FB_ECAT_DIAG(
	nEcMasterSlaveCount:= , 
	nEcMasterDevState:= , 
	nEcMasterDeviceId:= , 
	arrEcMasterNetId:= , 
	nEcMasterSlaveCountCfg:= , 
	wFrmXWcState:= , 
	bAllFrameWcStatesOK=> , 
	bEtherCATOK=> , 
	bFrameWcStateError=> , 
	bSlaveCountError=> , 
	bMasterDevStateError=> , 
	stMasterDevState=> , 
	bBusy=> , 
	bError=> , 
	iErrorID=> , 
	arrSlaveInfo:= arrEcatSlaveInfo);

IF nSlaveNr > iSLAVEADDR_ARR_SIZE THEN nSlaveNr := iSLAVEADDR_ARR_SIZE; END_IF
stSlaveInfo := arrEcatSlaveInfo[nSlaveNr];


FB_EVENTHANDLER(
	bClearAll:= bAckP, 
	bAlarmActive=> , 
	sEventText=> , 
	sEventSource=> , 
	sEventJson=> );

END_PROGRAM

// ---- POUs/MesTest.TcPOU
PROGRAM MesTest
VAR
	MES:						FB_MES_INTERFACE_V2;		(* Instance of MES-Interface function block *)
	bMES_InitOK					:BOOL := FALSE;
	RESP:						ST_REQUEST;				(* Reference to MES-Interface function block response *)
	RESET:						BOOL;					
	START:						BOOL;					
	STATE:						UDINT;
	INDEX:						INT;					
	
	COVER_BARCODE:				STRING:='288000060010020103725571';					(* COVER barcode *)
	COVER_PARENT:				STRING;					(* MRT parent barcode *)
	COVER_STATE:				ST_GET_OP_STATE;		(* Container of SFC State data which releated to Cover barcode *)
	COVER_INVENTORY:			ST_INVENTORY;			(* Result inventory of the import *)
	COVER_VALID:				BOOL;					
	
	CARRIER_BARCODE:			STRING:='288000000005020103725189';					(* CARRIER barcode *)
	CARRIER_PARENT:				STRING;					(* MRT parent barcode *)
	CARRIER_STATE:				ST_GET_OP_STATE;		(* Container of SFC State data which releated to Carrier barcode *)
	CARRIER_INVENTORY:			ST_INVENTORY;			(* Result inventory of the import *)
	CARRIER_VALID:				BOOL;					
	
	PCBA_BARCODE:				STRING:='380027351706990103944077';					(* 4010 PCBA barcode *)
	PCBA_PARENT:				STRING;					(* MRT parent barcode *)
	PCBA_STATE:					ST_GET_OP_STATE;		(* Container of SFC State data which releated to PCBA barcode *)
	PCBA_INVENTORY:				ST_INVENTORY;			(* Inventory data of PCBA *)
	PCBA_VALID:					BOOL;					
	PCBA_BOM:					ST_BOM;					(* Container of BOM releated to PCBA barcode *)
	PCBA_RECIPE:				STRING;
	PCBA_INVENTORY_LIST:		ST_INVENTORY_LIST;		(* Need to be filld with Inventory ID before try to assemble it *)
	PCBA_ASSY_RESULT:			E_TEST_STATE;			(* Assembly result Passed/Failed *)
	PCBA_CHECK_RESULT:			E_TEST_STATE;			(* Assembly result Passed/Failed *)
	PCBA_MATERIAL:				ST_MATERIAL;			(* Contains the PCBA material *)
	PCBA_SHOPORDER_LIST:		ST_SHOPORDER_LIST;		(* List of suitable sohoporder for the PCBA material *)
	
	FAN_BARCODE:				STRING:='288000000004000104014579';					(* FAN barcode *)
	FAN_PARENT:					STRING;					(* Parent of the FAN, need to be a PCBA barcode, with matching with BOM material. *)
	FAN_STATE:					ST_GET_OP_STATE;		(* Container of SFC State data which releated to Fan barcode *)
	FAN_INVENTORY:				ST_INVENTORY;			(* Result inventory of the import *)
	FAN_VALID:					BOOL;					
	
	MRT_BARCODE:				STRING;					(* MRT barcode *)
	MRT_STATE:					ST_GET_OP_STATE;		(* Container of SFC State data which releated to MRT barcode *)
	MRT_INVENTORY_LIST:			ST_INVENTORY_LIST;		(* Need to be filld with Inventory ID before try to assemble it *)
	MRT_ASSY_RESULT:			E_TEST_STATE;			(* Assembly result Passed/Failed *)
	MRT_BOM:					ST_BOM;					(* Container of BOM releated to PCBA barcode *)
	MRT_MATERIAL:				ST_MATERIAL;			(* Contains the MRT material *)
	MRT_MATERIAL_INFO:			ST_MATERIAL_INFO;		(* Contains the MRT material *)
	MRT_SHOPORDER_LIST:			ST_SHOPORDER_LIST;		(* List of suitable sohoporder for the MRT material *)
	
	(* Process variables *)		
	FAN_INSERT_CHECK_RESULT:		E_TEST_STATE;
	FAN_INSERT_CHECK_RECIPE:		STRING;
	
	FAN_CONNECTION_CEHCK_RESULT:	E_TEST_STATE;
	FAN_CONNECTION_CEHCK_RECIPE:	STRING;
	
	GAP_FILLER_CHECK_MRT_RESULT:	E_TEST_STATE;
	GAP_FILLER_CHECK_MRT_RECIPE:	STRING;
	GAP_FILLER_CHECK_COVER_RESULT:	E_TEST_STATE;
	GAP_FILLER_CHECK_COVER_RECIPE:	STRING;
	
	GAP_FILLER_RESULT:				E_TEST_STATE;
	GAP_FILLER_RECIPE:				STRING;
	
	SCREWING_RESULT:				E_TEST_STATE;
	SCREWING_RECIPE:				STRING;

	TestReceipeName					:String;
	TestCustomData					:String(1000);	
	(* Reusable variables*)
	(* Temporary containers for MES.GET_SHOPORDER_BY_MAT() *)

	SHOPORDER:					ST_SHOPORDER;
	RELEASE_COUNT:				STRING;
	
	(* Temporary containers for MES.VALIDATE_IN_BOM() *)
	COMPONENT_MATERIAL:			ST_MATERIAL;
	BOM_COMPONENT:				ST_BOM_COMPONENT;
	
	(*  *)
	MESDAT:						ST_MESDAT;
	NCDAT:						ST_MESDAT;
	
	
	DEBUG:						STRING;
	
	sRecipelist					:STRING(1000);
	sRecipe						:STRING;
	fbRecipeList				:FB_ReceipeList;
	bExecute					:BOOL;
END_VAR

IF bExecute THEN
	fbRecipeList(
		sReceipeListIn:= sRecipelist,
		sReceipeListOut=> sRecipelist,
		sReceipe=> sRecipe,
		bEmpty=> );
	bExecute := FALSE;
END_IF

//MRT_MATERIAL.MATERIAL:='00003981088'; 	//Preconfigured by the opreator
//MRT_MATERIAL.REVISION:='990';			//Preconfigured by the operator
RELEASE_COUNT:='1';						//Preconfigured by the operator - Required quantity.

IF bP1MesInitOK AND bP2MesInitOK AND NOT bMES_InitOK THEN
	IF MES.REMOTE_INIT_SERVICE() THEN
		bMES_InitOK := TRUE;
	END_IF
END_IF

CASE STATE OF
(* ###############################################################		Initialize		###########################################################################	*)
(*
	0:			(* Material setup based on the selected material *)
		IF MES.ASSY_GET_SHOPORDER_BY_MAT(MRT_MATERIAL, RELEASE_COUNT, INDEX, MRT_SHOPORDER_LIST) THEN
			STATE:=10;
		END_IF
	10: 		(* Slect ove suitable Shoporder - In this case work always with the idx:=0 *)
		IF MES.ASSY_GET_TOTAL_BOM_BY_SO(MRT_SHOPORDER_LIST.LIST[0].HANDLE, INDEX, MRT_BOM) THEN
			STATE:=100;
		END_IF
*)
(* ###############################################################		Wait for start	###########################################################################	*)
	100:		(* Wait the start trigger *)
		IF START THEN
			INDEX:=0;
			STATE:=30000;
			START:=FALSE;
		END_IF				
		
(* ################################################################################################################################################################
   #
   #
   #																	ST40-Automatic assembly
   #
   #
   ################################################################################################################################################################ *)
(* ##############################################################		MRT/Cover dispensing check 		###################################################################	*)
	30000:		(* Start OP_GAP_FILLER_CHECK in my case is index[0]. *)
		GAP_FILLER_CHECK_MRT_RESULT:=E_TEST_STATE.FAILED;
		INDEX:=0; // prepare the next operation
		IF MES.START_SFC(MRT_BARCODE, INDEX) THEN
			IF RESP.RESP_CODE='0' THEN
				STATE := STATE + 1;				//30010;
			ELSE
				DEBUG:='30000 - ASSY_START_SFC() failed with wrong rescode';
				STATE:=99999;
			END_IF
		END_IF

	30010: 		(* Get ricpe name *)
		IF MES.GET_RECIPE_NAME_BY_OPERATION_XML('OP_GAP_FILLER_CHECK_MRT', GAP_FILLER_CHECK_MRT_RECIPE) THEN
			IF GAP_FILLER_CHECK_MRT_RECIPE<>'' THEN
				STATE := STATE + 1;				// 30020;
			ELSE
				DEBUG:='30010 - ASSY_GET_RECIPE_NAME_BY_OPERATION() failed with wrong rescode or empty recipe';
				STATE:=99999;
			END_IF
		END_IF
		
	30020: 		(* Check dispensing quality... then set result. *)
		GAP_FILLER_CHECK_MRT_RESULT:=E_TEST_STATE.PASSED;
		STATE := STATE + 1;						//30030;	
		
	30030:		(* Complete OP_GAP_FILLER_CHECK in my case is index[4]. *)
		IF MES.COMPLETE_SFC(MRT_BARCODE, INDEX, GAP_FILLER_CHECK_MRT_RESULT) THEN
			IF RESP.RESP_CODE='0' THEN
				MRT_INVENTORY_LIST.LIST[1]:=COVER_INVENTORY;
				STATE := STATE + 1;				//30200;
			ELSE
				DEBUG:='30030 - ASSY_COMPLETE_SFC() failed with wrong rescode';
				STATE:=99999;
			END_IF
		END_IF

	30040:		(* Start OP_GAP_FILLER_CHECK in my case is index[4]. *)
		GAP_FILLER_CHECK_COVER_RESULT:=E_TEST_STATE.FAILED;
		INDEX:=1; // prepare the next operation
		IF MES.START_SFC(COVER_BARCODE, INDEX) THEN
			IF RESP.RESP_CODE='0' THEN
				STATE := STATE + 1;				//30010;
			ELSE
				DEBUG:='30000 - ASSY_START_SFC() failed with wrong rescode';
				STATE:=99999;
			END_IF
		END_IF

	30050: 		(* Get ricpe name *)
		IF MES.GET_RECIPE_NAME_BY_OPERATION_JSON('OP_GAP_FILLER_CHECK_COVER', GAP_FILLER_CHECK_COVER_RECIPE) THEN
			IF GAP_FILLER_CHECK_COVER_RECIPE<>'' THEN
				STATE := STATE + 1;				// 30020;
			ELSE
				DEBUG:='30010 - ASSY_GET_RECIPE_NAME_BY_OPERATION() failed with wrong rescode or empty recipe';
				STATE:=99999;
			END_IF
		END_IF
		
	30060: 		(* Check dispensing quality... then set result. *)
		GAP_FILLER_CHECK_COVER_RESULT:=E_TEST_STATE.PASSED;
		STATE := STATE + 1;						//30030;	
		
	30070:		(* Complete OP_GAP_FILLER_CHECK in my case is index[4]. *)
		IF MES.COMPLETE_SFC(COVER_BARCODE, INDEX, GAP_FILLER_CHECK_COVER_RESULT) THEN
			IF RESP.RESP_CODE='0' THEN
				MRT_INVENTORY_LIST.LIST[1]:=COVER_INVENTORY;
				STATE := STATE + 1;				//30200;
			ELSE
				DEBUG:='30030 - ASSY_COMPLETE_SFC() failed with wrong rescode';
				STATE:=99999;
			END_IF
		END_IF	

	30080:
			NCDAT.N := 1;
			NCDAT.MESDAT[NCDAT.N].RESPONSE_CODE := '4005';
			NCDAT.MESDAT[NCDAT.N].RESPONSE_DESCRIPTION := CONCAT('Camera error of POS#', INT_TO_STRING(2));
			NCDAT.MESDAT[NCDAT.N].CLIENT_DATE := fbP1MesInterface.GET_LOCAL_TIME();
			NCDAT.MESDAT[NCDAT.N].TEST_STATE := INT_TO_STRING(E_TEST_STATE.FAILED);
			NCDAT.MESDAT[NCDAT.N].TEST_STEP := INT_TO_STRING(NCDAT.N);
			NCDAT.MESDAT[NCDAT.N].VALUE := '0';
			STATE:=STATE + 10;

	30090:		(* Log NonConformance data *)
		IF MES.ASSY_SAVE_NCDAT(MRT_BARCODE, INDEX, NCDAT) THEN
			IF RESP.RESP_CODE = '0' THEN
				STATE:=STATE + 1;
			ELSE
				DEBUG:='30250 - SAVE_NCDAT() failed with wrong rescode';
				STATE:=99999;
			END_IF
		END_IF



	30100: 	(* Get MRT OP state 1026*)
			IF MES.GET_CURRENT_OPERATION_STATE(MRT_BARCODE,INDEX,MRT_STATE) THEN
				IF RESP.RESP_CODE = '0' THEN
					MRT_MATERIAL.MATERIAL := MRT_STATE.MAT_NO;
					MRT_MATERIAL.REVISION := MRT_STATE.REVISION;
					STATE:=STATE + 10;
				ELSE
					DEBUG:=' - Get op state MRT error';
					STATE:=99999;
				END_IF
			END_IF

	30110:
			IF MES.GET_MAT_CUSTOM_DATA(MRT_MATERIAL,INDEX) THEN		//1037
				IF RESP.RESP_CODE = '0' THEN
					STATE:=STATE + 10;
				ELSE
					DEBUG:=' - GET_MAT_CUSTOM_DATA error';
					STATE:=99999;
				END_IF
			END_IF
			
	30120:
			IF MES.GET_CUSTOM_DATA_BY_KEY(TestReceipeName,TestCustomData) THEN	//
				IF TestCustomData <> '' THEN
					STATE:=STATE + 1;
				ELSE
					DEBUG:=' - GET_CUSTOM_DATA_BY_KEY error';
					STATE:=99999;
				END_IF
			END_IF
			
			

			
(* ##############################################################		MRT final assembly 		###################################################################	*)
	30200:		(* Start OP_ASSY_AUTO_2 in my case is index[7]. *)
		INDEX:=2; // prepare the next operation, the inventory list is filled currently.
		IF MES.START_SFC(MRT_BARCODE, INDEX) THEN
			IF RESP.RESP_CODE='0' THEN
				STATE := STATE + 1;				//30210;
			ELSE
				DEBUG:='30200 - ASSY_START_SFC() failed with wrong rescode';
				STATE:=99999;
			END_IF
		END_IF
		
	30210: 		(* Assemble parts (PCBA and Cover into MRT) *)
		IF MES.ASSEMBLE_BY_INVENTORY_LIST(MRT_BARCODE, INDEX, MRT_INVENTORY_LIST) THEN
			IF RESP.RESP_CODE='0' THEN
				STATE := STATE + 1;						//30210;
				MRT_ASSY_RESULT:=E_TEST_STATE.PASSED;
			ELSE
				STATE := STATE + 2;						//30220; // jump to scrap
				MRT_ASSY_RESULT:=E_TEST_STATE.FAILED;
			END_IF
			
		END_IF	

	30220:		(* Scrap the PCBA if needed *)	
		IF MES.SCRAP_SFC(PCBA_BARCODE, INDEX) THEN
			DEBUG:='30220 - PCBA is scraped';
			STATE:=99999;
		END_IF
		
	30230:		(* Complete OP_ASSY_AUTO_2 in my case is index[7]. *)
		IF MES.COMPLETE_SFC(MRT_BARCODE, INDEX, MRT_ASSY_RESULT) THEN
			IF RESP.RESP_CODE='0' THEN
				STATE:=100;						//40000;
			ELSE
				DEBUG:='30230 - ASSY_COMPLETE_SFC() failed with wrong rescode';
				STATE:=99999;
			END_IF
		END_IF
		

END_CASE
FB_CALL_ACT();;

ACTION FB_CALL_ACT:
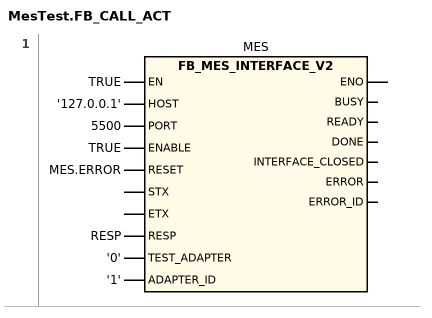
// NETWORK 1
MES(
    HOST := '127.0.0.1',
    PORT := 5500,
    ENABLE := TRUE,
    RESET := MES.ERROR,
    RESP := RESP,
    TEST_ADAPTER := '0',
    ADAPTER_ID := '1'); // FB_MES_INTERFACE_V2
END_ACTION

END_PROGRAM

// ---- POUs/FBs/FB_ReceipeList.TcPOU
FUNCTION_BLOCK FB_ReceipeList
VAR_INPUT
	sReceipeListIn			:STRING(1000);
END_VAR
VAR_OUTPUT
	sReceipeListOut			:STRING(1000);
	sReceipe				:STRING;
	bEmpty					:BOOL;
END_VAR
VAR
	nPosition				:INT;
END_VAR

nPosition := FIND(sReceipeListIn,';');
IF nPosition > 0 THEN
	sReceipe := LEFT(sReceipeListIn,(nPosition - 1));
	sReceipeListOut	:= DELETE(sReceipeListIn,(nPosition + 1),0);
ELSE
	sReceipe := sReceipeListIn;
	sReceipeListOut	:= '';
END_IF
bEmpty := (LEN(sReceipeListOut) <= 0);

END_FUNCTION_BLOCK

// ---- POUs/FBs/FB_Door.TcPOU
FUNCTION_BLOCK FB_Door
VAR_INPUT
	bDoorButton			:BOOL;			// Ajtó gomb benemet
	bOpenEnable			:BOOL;			// Ajtó nyitást lehetséges folyamat oldalról
	bDoorsClosed		:BOOL;			// Ajtók becsukva
	bDoorsLocked		:BOOL;			// Ajtók reteszelve
	bBlink				:BOOL;			// Ajtó led villogtatáshoz külső blinker
END_VAR
VAR_OUTPUT
	bCloseOut			:BOOL;			// Ajtó zárás kimenet
	bDoorButtonLED		:BOOL;			// Ajtó gomb LED kimenet
	bObenRequestOut		:BOOL;			// Ajtó nyitás kérés kimenet a körasztalnak
END_VAR
VAR
	rtDoorButton		:R_Trig;		// Ajtó gombnyomás felfutó él
	rsOpenRequest		:RS;			// Nyitás igény rögzítés
	tOpenForce			:TON;			// Nyitás kényszerítés időzítő
	tOpenForceDelay		:TIME := T#5S;	// Nyitás kényszerítés késleltetés
	ftDoorsLocked		:F_Trig;		// Ajtó retelszelve lefutó él
END_VAR

(* Ajtó kezelő FB működés:
Zárás: csukva vannak az ajtók és gombnyomás történik
Nyitás esetek (ha reteszelve vannak az ajtók és gombnyomás történik):
	1. Nyitás: ha a folyamat engedélyt ad a nyitásra
	2. Nyitás igény rögzítés: ha a folyamat nem ad engedélyt a nyitásra, 
		innen mehet 1.-be, vagy 3.-ba, vagy ismételt gombnyomásra törli az igényt
	3. Kényszerített nyitás: ha 5 másodpercig nyomják a gombot, mindenképp kinyit *)

// Ajtó gomb felfutó él képzés
rtDoorButton(CLK:= bDoorButton);

// Zárás
IF rtDoorButton.Q AND bDoorsClosed AND NOT bDoorsLocked THEN
	bCloseOut := TRUE;
END_IF

// Nyitás kérés
rsOpenRequest(
	SET:= rtDoorButton.Q AND bDoorsClosed AND bDoorsLocked, 
	RESET1:= NOT bDoorsLocked OR (rtDoorButton.Q AND rsOpenRequest.Q1),  
	Q1=> bObenRequestOut
	);

// Kényszerített nyitás
tOpenForce(IN:= bDoorButton AND bDoorsLocked, PT:= tOpenForceDelay);

// Nyitás kimenet
IF (rsOpenRequest.Q1 AND bOpenEnable) 
	OR tOpenForce.Q
	OR ftDoorsLocked.Q
THEN
	bCloseOut := FALSE;
END_IF

// Ajtó gomb LED vezérlés
IF bDoorsLocked THEN
	IF rsOpenRequest.Q1 THEN
		bDoorButtonLED := bBlink;
	ELSE
		bDoorButtonLED := TRUE;
	END_IF
ELSE
	bDoorButtonLED := FALSE;
END_IF

// Ajtó retelszelve lefutó él
ftDoorsLocked(CLK:= bDoorsLocked, Q=> );

END_FUNCTION_BLOCK

// ---- POUs/FBs/FB_WorkLight.TcPOU
FUNCTION_BLOCK FB_WorkLight
VAR_INPUT
	bDoorClose					:BOOL;
	bManualCtrl					:BOOL;
	nEcoTime					:UINT := 5;
END_VAR
VAR_OUTPUT
	bLightCtrl					:BOOL;
END_VAR
VAR
	tEcoTime					:TON;
	rtDoorOn					:R_Trig;
	rtManualOn					:R_Trig;
	rtDoorOff					:R_Trig;
	rtManualOff					:R_Trig;
	rtTimerOff					:R_Trig;
END_VAR

rtDoorOn(CLK:= NOT bDoorClose);
rtManualOn(CLK:= bManualCtrl);
rtDoorOff(CLK:= bDoorClose);
rtManualOff(CLK:= NOT bManualCtrl);
rtTimerOff(CLK:= tEcoTime.Q);
tEcoTime(IN:= bLightCtrl, PT:= (nEcoTime * T#1M));

IF rtDoorOn.Q OR rtManualOn.Q THEN
	bLightCtrl := TRUE;
	bManualCtrl := TRUE;
END_IF

IF rtDoorOff.Q OR rtManualOff.Q OR rtTimerOff.Q THEN
	bLightCtrl := FALSE;
	bManualCtrl := FALSE;
END_IF

END_FUNCTION_BLOCK

// ---- POUs/FBs/FB_BISM.TcPOU
FUNCTION_BLOCK FB_BISM
(*Ez az FB BIS M-458-045-001-07-S4-el lett tesztelve.
TAG: BIS M-191-02/A UID 8 byte read only, User data 2000 byte.
Saját adatot írtunk a TAG-ekbe 1..255ig és nem a UID-t olvasunk ki, hanem user data-t.
Ezt a BISM 458 konfigjában be kell állítani: Activity at tag present -> Send data*)

VAR_INPUT
	sName				:STRING; (*Olvasó neve, HMI*)
	bReset				:BOOL;	(*Software reset*)
	bHeadOff			:BOOL;	(*Antenna lekapcsolása*)
END_VAR
VAR_OUTPUT
	bTagPresent			:BOOL;
	//nTAGData			:ULINT; (*Data which was read from the data carrier*)
	nTAGData			:BYTE;
	sTAGData			:STRING;
	nErrorCode			:BYTE; (*Error code when AF = 1*)
END_VAR
VAR
	InData				AT %I* :ARRAY[0..9] OF BYTE;
	bBB					:BOOL; (*Power: 1 = Device ready, 0 = Device in groung state*)
	bHF					:BOOL; (*Head failure: 1 = Head is turned off, 0 = Head is turned on*)
	bAF					:BOOL; (*Job error: 1 = Job incorrectly processed, 0 = Job processed without errors*)
	bAE					:BOOL; (*Job end: 1 = Job processed without errors, 0 = No job or job running*)
	bAA					:BOOL; (*Job accepted: 1 = Job accepted, 0 = No job*)
	bCP					:BOOL; (*Codetag present: 1 = Data carrier is within range of the head, 0 = no data carrier*)
	
	OutData				AT %Q* :ARRAY[0..9] OF BYTE;
	bTI					:BOOL; (*Toggle bit: State change during job*)	
	bKA					:BOOL; (*Head on/off: 1 = Head on, 0 = Head off*)
	bGR					:BOOL; (*Basic state: 1 = Software reset, 0 = Normal operation*)
	bAV					:BOOL; (*Job: 1 = New job, 0 = No new job*)
	
	(*User data íráshoz*)
	nCommandDesignator	:BYTE := 50; (*50 = write*)
	nNbrOfBytes			:BYTE := 1; (*1 byteot írunk*)
	(*User data íráshoz, HMI-ről írjuk be*)
	nWriteValue			:BYTE; (*Beírt érték*)
	bWriteCmd			:BOOL; 	
END_VAR

bBB := InData[0].7;
bHF := InData[0].6;
bAF := InData[0].3;
bAE := InData[0].2;
bAA := InData[0].1;
bCP := InData[0].0;

IF bAF THEN 
	nErrorCode := InData[1];
	nTAGData := 0;
ELSE 
	IF bCP THEN
		//nTAGData :=	InData[1];
		nTAGData := ULINT_TO_BYTE(
					SHL(BYTE_TO_ULINT(InData[8] AND 127), 56) +
					SHL(BYTE_TO_ULINT(InData[7]), 48) +
					SHL(BYTE_TO_ULINT(InData[6]), 40) +
					SHL(BYTE_TO_ULINT(InData[5]), 32) +
					SHL(BYTE_TO_ULINT(InData[4]), 24) +
					SHL(BYTE_TO_ULINT(InData[3]), 16) +
					SHL(BYTE_TO_ULINT(InData[2]), 8) +
					InData[1]);		
	ELSE 
		nTAGData := 0;
	END_IF
	IF bBB THEN
		nErrorCode := 0;
	ELSE 
		nErrorCode := 255;
	END_IF
END_IF

bTagPresent := bCP;
//sTAGData := ULINT_TO_STRING(nTAGData);
sTAGData := BYTE_TO_STRING(nTAGData);

bGR := bReset;
bKA := bHeadOff;
OutData[0].0 := bAV;
OutData[0].2 := bGR;
OutData[0].5 := bKA;
OutData[0].6 := bTI;
OutData[9] := OutData[0];

(*Íráshoz*)
bAV := bWriteCmd;
OutData[1] := nCommandDesignator;
OutData[2] := 0; (*Start address*)
OutData[4] := nNbrOfBytes;
OutData[6] := nWriteValue;
IF bWriteCmd AND bAE THEN
	bWriteCmd := FALSE;
END_IF

END_FUNCTION_BLOCK

// ---- POUs/FBs/FB_FullCycleTime.TcPOU
FUNCTION_BLOCK FB_FullCycleTime
VAR_INPUT
	bPalletSensor			:BOOL;
	timTimeMax				:TIME:= T#120S;
END_VAR
VAR_OUTPUT
	nCurrentCycleTime		:REAL;
	arrCycleTimes			:ARRAY [1..10] OF REAL;
END_VAR
VAR
	tCycleTime				:TON;
	rStart					:R_TRIG;
END_VAR

rStart(CLK:= bPalletSensor);
tCycleTime(IN:= TRUE, PT:= timTimeMax);

IF 		rStart.Q THEN
				MEMMOVE(ADR(arrCycleTimes)+4,ADR(arrCycleTimes),SIZEOF(arrCycleTimes)-4);
				arrCycleTimes[1] := nCurrentCycleTime;
				tCycleTime(IN:= FALSE);
ELSIF	NOT tCycleTime.Q THEN
				nCurrentCycleTime := (TIME_TO_REAL(tCycleTime.ET) / 1000);
ELSE
				nCurrentCycleTime := (TIME_TO_REAL(timTimeMax) / 1000);
END_IF

END_FUNCTION_BLOCK

// ---- POUs/FBs/FB_KRC4.TcPOU
FUNCTION_BLOCK FB_KRC4
VAR_INPUT
	sName				:STRING;
	bEn					:BOOL;				(* Engedély jel *)
	bZoneEnable			:BOOL;				(* Zóna engedély *)
	bAutoCycle			:BOOL;				(* Automa teljes ciklus *)	
	bExecuteProg		:BOOL;				(* Csakegy program végrehajtása *)
	nProgNr				:BYTE;				(* Program szám *)
	timBaseState		:TIME:=T#15S;		(* Alaphelyzet felvételi idő*)
	bAck				:BOOL; 				(* Hibanyugta *)
	stEventArray		:ARRAY [0..7] OF TcEventEntry;		(* Event array definition *)
END_VAR
VAR_OUTPUT
	bReady				:BOOL;				(* Folyamat üzemkész *)
	bBusy				:BOOL;				(* Folyamat aktív *)
	bDone				:BOOL;				(* Folyamat kész *)
	bPendantMode		:BOOL;				(* Teach pendant mód aktív *)
	bError				:BOOL;				(* Hiba bit*)
	sError				:STRING(255);		(* Hiba string*)
END_VAR
VAR
	tBaseState			:TON;
	RobotIn				:U_KRC_Input;
	RobotOut			:U_KRC_Output;
	bErrNotReady		:BOOL;
	bErrBaseTimeout		:BOOL;
	nState				:UDINT;
	nStateLast			:UDINT;
	sState				:STRING;
	aErrorDesc			:ARRAY [0..7] OF STRING := [
	' Kuka KRC rendszerhiba : - Információ a "pendant"-on ', 
	' Kuka KRC programhiba : - A kiválasztott program nem hajtható végre ', 
	' Kuka KRC  pozícióhiba : - A kiválasztott pozíció nem elérhető ', 
	' Kuka KRC  paraméterhiba : - Hibás paraméter ', 
	' Kuka KRC  vákuumhiba : - A vákuum nem épült fel ', 
	' Kuka KRC  darabvesztés hiba : - A vákuumfejről leesett az alkatrész ',
	' Kuka KRC  üzemzavar : - Üzem közben a "Ready" jel megszűnt ',
	' Kuka KRC  üzemzavar : - A robot nem tud alaphelyzetbe mozogni '];
	sEmpty				:STRING:='';
	bIsInitalized		:BOOL;
	fbAlarmArray		:ARRAY [0..7] OF FB_TcAlarm;
	arrAlarms			:ARRAY [0..7] OF BOOL;
	i					:INT;
END_VAR

(*Időzítők***************************************************)
tBaseState(IN:= (nState > 0 AND nState < 10000), PT:= timBaseState);
(*Triggerek**************************************************)

(*Hibakezelés************************************************)
IF nState >= 120 AND nState < 150000 AND NOT RobotIn.Status.bReady THEN
	bErrNotReady := TRUE;
END_IF
IF tBaseState.Q AND NOT bErrBaseTimeout THEN
	bErrBaseTimeout := TRUE;
END_IF

bError := (nState > 10000) AND	(NOT RobotIn.Status.bAlarm OR
							RobotIn.Status.bProgramError OR
							RobotIn.Status.bPositionError OR
							RobotIn.Status.bParameterError OR
							RobotIn.Status.bVacuumError OR
							RobotIn.Status.bWorpieceError OR 
							bErrNotReady OR
							bErrBaseTimeout);

arrAlarms[0] := NOT RobotIn.Status.bAlarm;
arrAlarms[1] := RobotIn.Status.bProgramError;
arrAlarms[2] := RobotIn.Status.bPositionError;
arrAlarms[3] := RobotIn.Status.bParameterError;
arrAlarms[4] := RobotIn.Status.bVacuumError;
arrAlarms[5] := RobotIn.Status.bWorpieceError;
arrAlarms[6] := bErrNotReady;
arrAlarms[7] := bErrBaseTimeout;

					
IF nState > 0 AND nState < 150000 THEN
	nStateLast := nState;
	IF	bError THEN
			nState := 200000;
	END_IF
END_IF

(*Pendant mód ************************************************)
bPendantMode := RobotIn.Status.bT1 OR RobotIn.Status.bT2;
IF bPendantMode THEN
	nState := 150000;
END_IF

(*Engedélyek *************************************************)
IF 	(NOT bEn AND NOT bPendantMode) OR								// nincs engedély, és pendantról sem szeretnék használni
	(NOT RobotIn.Status.bUserSAF AND NOT bPendantMode) THEN			// nincs ajtókör, és pendantról sem szeretnék használni
		nState := 0;
END_IF
RobotOut.Control.bEnableMoveInPalettZone := RobotIn.Status.bReqMoveInPalettZone AND bZoneEnable;

(*Automata üzem *********************************************)
CASE nState OF
	0:		sState := CONCAT(UDINT_TO_STRING(nState) ,' - Vészkör vagy ajtókör bontva - Működtetések törlése');
			RobotOut.Control.bPgnoParity := FALSE;
			RobotOut.Control.bPgnoValid := FALSE;
			RobotOut.Control.bExtStart := FALSE;
			RobotOut.Control.bMoveEnable := FALSE;
			RobotOut.Control.bConfMess := FALSE;
			RobotOut.Control.bDrivesOff := FALSE;
			RobotOut.Control.bDrivesOn := FALSE;
			RobotOut.Control.bIOAct := FALSE;
			RobotOut.Control.bVacuumErrorClear := FALSE;
			bErrNotReady := FALSE;
			bErrBaseTimeout := FALSE;
			bReady := FALSE;
			bBusy := FALSE;	
			IF	bEn AND
				RobotIn.Status.bAlarm AND
				RobotIn.Status.bIntEStop AND
				RobotIn.Status.bUserSAF THEN
					bBusy := TRUE;
					nState := nState + 20;
			END_IF
			
	20:		sState := CONCAT(UDINT_TO_STRING(nState) ,' - Alaphelyzetfelvétel - "STOP_MESS" ellenőrzése');
			IF RobotIn.Status.bStopMess THEN
				RobotOut.Control.bMoveEnable := TRUE;
				nState := nState + 20;
			END_IF

	40:		sState := CONCAT(UDINT_TO_STRING(nState) ,' - Alaphelyzetfelvétel - "DRIVES_ON"');
			RobotOut.Control.bDrivesOn := TRUE;
			IF RobotIn.Status.bPeriReday THEN
				RobotOut.Control.bDrivesOn := FALSE;
				nState := nState + 20;
			END_IF

	60:		sState := CONCAT(UDINT_TO_STRING(nState) ,' - Alaphelyzetfelvétel - "CONF_MESS"');
			RobotOut.Control.bConfMess := TRUE;
			IF NOT RobotIn.Status.bStopMess THEN
				RobotOut.Control.bConfMess := FALSE;
				nState := nState + 20;
			END_IF

	80:		sState := CONCAT(UDINT_TO_STRING(nState) ,' - Alaphelyzetfelvétel - "EXT_START"');
			RobotOut.Control.bExtStart := TRUE;
			IF RobotIn.Status.bPgnoReq THEN
				RobotOut.Control.bExtStart := FALSE;
				nState := nState + 20;
			END_IF

	100:	sState := CONCAT(UDINT_TO_STRING(nState) ,' - Alaphelyzetfelvétel - "Home" program betöltése');
			RobotOut.Control.nProgNr := 1;
			IF RobotIn.Status.nProgNr = RobotOut.Control.nProgNr THEN
				RobotOut.Control.bPgnoParity := TRUE;
				RobotOut.Control.bPgnoValid := TRUE;
				nState := nState + 20;
			END_IF

	120:	sState := CONCAT(UDINT_TO_STRING(nState) ,' - Alaphelyzetfelvétel - várakozás "Home" program indítására');
			IF RobotIn.Status.bApplRun THEN
				RobotOut.Control.bPgnoParity := FALSE;
				RobotOut.Control.bPgnoValid := FALSE;
				nState := nState + 20;
			END_IF

	140:	sState := CONCAT(UDINT_TO_STRING(nState) ,' - Alaphelyzetfelvétel - várakozás "Home" program befejezésére');
			IF NOT RobotIn.Status.bApplRun THEN
				nState := nState + 20;
			END_IF
		
	160:	nState := 10000;

(* Alaphelyzet *********************************************************************)
	10000:	sState := CONCAT(UDINT_TO_STRING(nState) ,' - Alaphelyzet - Várakozás parancsra');
			IF		bAutoCycle AND NOT bExecuteProg THEN							// Automata ciklus kérés
						bReady := TRUE;
						bBusy := TRUE;
						bDone := FALSE;
						nState := 11000;
			ELSIF	NOT bAutoCycle AND bExecuteProg THEN							// Egyszeri program végrehajtás
						bReady := TRUE;
						bBusy := TRUE;
						bDone := FALSE;
						nState := 12000;
			ELSIF	NOT bAutoCycle AND NOT bExecuteProg THEN						// Nincs parancs
						bReady := TRUE;
						bBusy := FALSE;
						bDone := FALSE;		
			END_IF

	(*-----=== Teljes automata ciklus ===-----*)
	11000:	sState := CONCAT(UDINT_TO_STRING(nState) ,' - "PCBA felvétel" 10. program betöltése');
			RobotOut.Control.nProgNr := 10;
			IF RobotIn.Status.nProgNr = RobotOut.Control.nProgNr THEN
				RobotOut.Control.bPgnoParity := TRUE;
				RobotOut.Control.bPgnoValid := TRUE;
				nState := nState + 20;
			END_IF

	11020:	sState := CONCAT(UDINT_TO_STRING(nState) ,' - "PCBA felvétel" 10. program indítására');
			IF RobotIn.Status.bApplRun THEN
				RobotOut.Control.bPgnoParity := FALSE;
				RobotOut.Control.bPgnoValid := FALSE;
				nState := nState + 20;
			END_IF

	11040:	sState := CONCAT(UDINT_TO_STRING(nState) ,' - Várakozás "PCBA felvétel" 10. program befejezésére');
			IF NOT RobotIn.Status.bApplRun THEN
				nState := nState + 20;
			END_IF			

	11060:	sState := CONCAT(UDINT_TO_STRING(nState) ,' - "PCBA behelyezése" 11. program betöltése');
			RobotOut.Control.nProgNr := 11;
			IF RobotIn.Status.nProgNr = RobotOut.Control.nProgNr THEN
				RobotOut.Control.bPgnoParity := TRUE;
				RobotOut.Control.bPgnoValid := TRUE;
				nState := nState + 20;
			END_IF

	11080:	sState := CONCAT(UDINT_TO_STRING(nState) ,' - "PCBA behelyezése" 11. program indítására');
			IF RobotIn.Status.bApplRun THEN
				RobotOut.Control.bPgnoParity := FALSE;
				RobotOut.Control.bPgnoValid := FALSE;
				nState := nState + 20;
			END_IF

	11100:	sState := CONCAT(UDINT_TO_STRING(nState) ,' - Várakozás "PCBA behelyezése" 11. program befejezésére');
			IF NOT RobotIn.Status.bApplRun THEN
				nState := nState + 20;
			END_IF				

	11120:	sState := CONCAT(UDINT_TO_STRING(nState) ,' - "Cover felvétel" 12. program betöltése');
			RobotOut.Control.nProgNr := 12;
			IF RobotIn.Status.nProgNr = RobotOut.Control.nProgNr THEN
				RobotOut.Control.bPgnoParity := TRUE;
				RobotOut.Control.bPgnoValid := TRUE;
				nState := nState + 20;
			END_IF

	11140:	sState := CONCAT(UDINT_TO_STRING(nState) ,' - "Cover felvétel" 12. program indítására');
			IF RobotIn.Status.bApplRun THEN
				RobotOut.Control.bPgnoParity := FALSE;
				RobotOut.Control.bPgnoValid := FALSE;
				nState := nState + 20;
			END_IF

	11160:	sState := CONCAT(UDINT_TO_STRING(nState) ,' - Várakozás "Cover felvétel" 12. program befejezésére');
			IF NOT RobotIn.Status.bApplRun THEN
				nState := nState + 20;
			END_IF			

	11180:	sState := CONCAT(UDINT_TO_STRING(nState) ,' - "Cover behelyezése" 13. program betöltése');
			RobotOut.Control.nProgNr := 13;
			IF RobotIn.Status.nProgNr = RobotOut.Control.nProgNr THEN
				RobotOut.Control.bPgnoParity := TRUE;
				RobotOut.Control.bPgnoValid := TRUE;
				nState := nState + 20;
			END_IF

	11200:	sState := CONCAT(UDINT_TO_STRING(nState) ,' - "Cover behelyezése" 13. program indítására');
			IF RobotIn.Status.bApplRun THEN
				RobotOut.Control.bPgnoParity := FALSE;
				RobotOut.Control.bPgnoValid := FALSE;
				nState := nState + 20;
			END_IF

	11220:	sState := CONCAT(UDINT_TO_STRING(nState) ,' - Várakozás "Cover behelyezése" 13. program befejezésére');
			IF NOT RobotIn.Status.bApplRun THEN
				nState := nState + 20;
			END_IF

	11240:	sState := CONCAT(UDINT_TO_STRING(nState) ,' - Várakozás indítójel törlésére');
			bBusy := FALSE;
			bDone := TRUE;
			IF NOT bAutoCycle THEN
				bDone := FALSE;
				nState := 10000;
			END_IF

	(*-----=== Egy program végrehajtása ===-----*)
	12000:	sState := CONCAT(UDINT_TO_STRING(nState) ,CONCAT(' - ',CONCAT(BYTE_TO_STRING(nProgNr),'. program betöltése')));
			RobotOut.Control.nProgNr := nProgNr;
			IF RobotIn.Status.nProgNr = RobotOut.Control.nProgNr THEN
				RobotOut.Control.bPgnoParity := TRUE;
				RobotOut.Control.bPgnoValid := TRUE;
				nState := nState + 20;
			END_IF

	12020:	sState := CONCAT(UDINT_TO_STRING(nState) ,CONCAT(' - ',CONCAT(BYTE_TO_STRING(nProgNr),'. program indítása')));
			IF RobotIn.Status.bApplRun THEN
				RobotOut.Control.bPgnoParity := FALSE;
				RobotOut.Control.bPgnoValid := FALSE;
				nState := nState + 20;
			END_IF

	12040:	sState := CONCAT(UDINT_TO_STRING(nState) ,CONCAT(' - Várakozás a ',CONCAT(BYTE_TO_STRING(nProgNr),'. program befejezésére')));
			IF NOT RobotIn.Status.bApplRun THEN
				nState := nState + 20;
			END_IF			

	12060:	sState := CONCAT(UDINT_TO_STRING(nState) ,' - Várakozás indítójel törlésére');
			bBusy := FALSE;
			bDone := TRUE;
			IF NOT bExecuteProg THEN
				bDone := FALSE;
				nState := 10000;
			END_IF

(* Pendant mód *********************************************************************)
	150000:	sState := CONCAT(UDINT_TO_STRING(nState) ,' - Pendant mód');
			IF NOT bPendantMode THEN
				nState := 0;
			ELSE
				RobotOut.Control.bPgnoParity := FALSE;
				RobotOut.Control.bPgnoValid := FALSE;
				RobotOut.Control.bExtStart := FALSE;
				RobotOut.Control.bMoveEnable := TRUE;
				RobotOut.Control.bConfMess := FALSE;
				RobotOut.Control.bDrivesOff := FALSE;
				RobotOut.Control.bDrivesOn := FALSE;
				RobotOut.Control.bIOAct := FALSE;
				RobotOut.Control.bVacuumErrorClear := FALSE;	
			END_IF
			
(* Hibakezelés *********************************************************************)
	200000:	sState := CONCAT(UDINT_TO_STRING(nState) ,CONCAT(' - Hiba, ebből az állapotból: ' ,sState));
			RobotOut.Control.bPgnoParity := FALSE;
			RobotOut.Control.bPgnoValid := FALSE;
			RobotOut.Control.bExtStart := FALSE;
			RobotOut.Control.bMoveEnable := FALSE;
			RobotOut.Control.bConfMess := FALSE;
			RobotOut.Control.bDrivesOff := FALSE;
			RobotOut.Control.bDrivesOn := FALSE;
			RobotOut.Control.bIOAct := FALSE;
			RobotOut.Control.bVacuumErrorClear := FALSE;
			bReady := FALSE;
			bBusy := FALSE;	
			nState := nState + 20;

(* Hibakezelés *********************************************************************)
	200020:	IF bAck THEN
				bErrNotReady := FALSE;
				bErrBaseTimeout := FALSE;
				FOR i:=0 TO 7 DO
					IF fbAlarmArray[i].eConfirmationState = 2 THEN
						fbAlarmArray[i].Confirm(0);
					END_IF
				END_FOR					
				nState := nState + 20;
			END_IF
			
	200040:	sState := CONCAT(UDINT_TO_STRING(nState) ,' - Hibatörlés - "STOP_MESS" ellenőrzése');
			IF RobotIn.Status.bStopMess THEN
				RobotOut.Control.bMoveEnable := TRUE;
				nState := nState + 20;
			END_IF

	200060:	sState := CONCAT(UDINT_TO_STRING(nState) ,' - Hibatörlés - "DRIVES_ON"');
			RobotOut.Control.bDrivesOn := TRUE;
			IF RobotIn.Status.bPeriReday THEN
				RobotOut.Control.bDrivesOn := FALSE;
				nState := nState + 20;
			END_IF

	200080:	sState := CONCAT(UDINT_TO_STRING(nState) ,' - Hibatörlés - "CONF_MESS"');
			RobotOut.Control.bConfMess := TRUE;
			IF NOT RobotIn.Status.bStopMess THEN
				RobotOut.Control.bConfMess := FALSE;
				nState := nState + 20;
			END_IF
	
	200100:	sState := CONCAT(UDINT_TO_STRING(nState) ,' - Alaphelyzetfelvétel - "EXT_START"');
			RobotOut.Control.bExtStart := TRUE;
			IF RobotIn.Status.bPgnoReq THEN
				RobotOut.Control.bExtStart := FALSE;
				nState := 100;
			END_IF
ELSE
	sState := CONCAT(UDINT_TO_STRING(nState) ,' - Nem használt állapot');
END_CASE	


(*Hiba string*)
IF bError THEN
	sError := sName;
	FOR i:=0 TO 7 DO
		IF arrAlarms[i] THEN
			sError :=  CONCAT(sError, aErrorDesc[i]);
			IF (fbAlarmArray[i].eConfirmationState <> 2 AND fbAlarmArray[i].nTimeCleared <> 0 AND fbAlarmArray[i].nTimeConfirmed <> 0) OR //Ha már volt alarm, akkor van bennük érték
				(fbAlarmArray[i].eConfirmationState = 1 AND fbAlarmArray[i].nTimeCleared = 0 AND fbAlarmArray[i].nTimeConfirmed = 0)	//Első futás esetén
			THEN
				fbAlarmArray[i].Raise(0);
			END_IF
		END_IF
	END_FOR 
ELSE
	sError := sEmpty;
END_IF

(*Hiba kezelés Tc3_EventLogger*)
IF NOT bIsInitalized THEN
	bIsInitalized := TRUE;
	FOR i:=0 TO 7 DO
		fbAlarmArray[i].CreateEx(stEventArray[i], TRUE, 0);
	END_FOR
END_IF

(*Hiba törlés (nyugtázott és megszűnt)*)
FOR i:=0 TO 7 DO
	IF fbAlarmArray[i].eConfirmationState = 3 AND NOT bError THEN
		fbAlarmArray[i].Clear(0, FALSE);
	END_IF
END_FOR

END_FUNCTION_BLOCK

// ---- POUs/FBs/FB_Conveyor.TcPOU
FUNCTION_BLOCK FB_Conveyor
VAR_INPUT
	sName					:STRING;
	bEn						:BOOL;				(*Enable - Engedély jel*)
	bEHA					:BOOL; 				(*Error-handling active - Hibafigyelés aktív*)
	bDisableManualCmd		:BOOL;				(*Manual control disable*)
	bConveyorOnL			:BOOL;				(*Control to Motor on - vezérlés parancs motor indításhoz*)
	bConveyorOnR			:BOOL;				(*Control to Motor on - vezérlés parancs motor indításhoz*)
	timReset				:TIME := T#2S;		(*Resettime - Hibatörlési idő*)
	bAck					:BOOL; 				(*Acknowledge - Hibanyugta*)
	i_bConveyorOK	AT %I*	:BOOL;				(*Conveyor drive OK - motorindító üzemkész*)
	stStartEvent			:TcEventEntry;		(*Event definition*)
	stRunEvent				:TcEventEntry;		(*Event definition*)
END_VAR
VAR_OUTPUT
	bMotorOn				:BOOL;				(* Motor on - Motor bekapcsolva *)
	bError					:BOOL;				(* Error bit - Hiba van *)
	sError					:STRING(255);		(* Error string - Hiba string *)
	q_bConveyorOnL	AT %Q*	:BOOL;				(* Motor on signal - Motor vezérlés bekapcsolása*)
	q_bConveyorOnR	AT %Q*	:BOOL;				(* Motor on signal - Motor vezérlés bekapcsolása*)
	q_bConveyorRst	AT %Q*	:BOOL;				(* Motor reset signal - Motor hibatörlés*)
END_VAR
VAR
	tMotorOn			:TON;
	tError,tFault		:TON;
	tReset				:TON;
	bErrOn,bErrRun		:BOOL;
	aErrorDesc			:ARRAY [0..1] OF STRING := [
	' motor hiba : a motorvezérlő nem indítható ', 
	' motor hiba : a motorvezérlő hibába van '];
	sEmpty				:STRING:='';
	bIsInitalized		:BOOL;
	fbStartAlarm		:FB_TcAlarm;
	fbRunAlarm			:FB_TcAlarm;
END_VAR

(*Hibanyugta*)
IF bAck OR NOT(bEHA) THEN
	bErrOn:=FALSE;
	bErrRun:=FALSE;
END_IF;

(* Motor bekapcsolási hiba *)
IF bEn AND bEHA AND (q_bConveyorOnL OR q_bConveyorOnR) AND NOT i_bConveyorOK THEN
	bErrOn:=TRUE;
	IF (fbStartAlarm.eConfirmationState <> 2 AND fbStartAlarm.nTimeCleared <> 0 AND fbStartAlarm.nTimeConfirmed <> 0) OR //Ha már volt alarm, akkor van bennük érték
		(fbStartAlarm.eConfirmationState = 1 AND fbStartAlarm.nTimeCleared = 0 AND fbStartAlarm.nTimeConfirmed = 0)	//Első futás esetén
	THEN
		fbStartAlarm.Raise(0);
	END_IF
END_IF;

(* Motor üzemzavar *)
tFault(IN:= bEn AND bEHA AND NOT i_bConveyorOK AND NOT bErrRun, PT:= T#5S);
IF tFault.Q THEN
	bErrRun:=TRUE;
	IF (fbRunAlarm.eConfirmationState <> 2 AND fbRunAlarm.nTimeCleared <> 0 AND fbRunAlarm.nTimeConfirmed <> 0) OR //Ha már volt alarm, akkor van bennük érték
		(fbRunAlarm.eConfirmationState = 1 AND fbRunAlarm.nTimeCleared = 0 AND fbRunAlarm.nTimeConfirmed = 0)	//Első futás esetén
	THEN
		fbRunAlarm.Raise(0);
	END_IF
END_IF;

(* Hibagyűjtő *)
bError := bErrOn OR bErrRun;

(*Vezérlés*)
IF 		bEn AND bConveyorOnL AND NOT bConveyorOnR AND i_bConveyorOK AND (NOT(bEHA) OR NOT(bError)) THEN
			q_bConveyorOnL := TRUE;
			q_bConveyorOnR := FALSE;
ELSIF	bEn AND NOT bConveyorOnL AND bConveyorOnR AND i_bConveyorOK AND (NOT(bEHA) OR NOT(bError)) THEN
			q_bConveyorOnL := FALSE;
			q_bConveyorOnR := TRUE;
ELSE
	q_bConveyorOnL := FALSE;
	q_bConveyorOnR := FALSE;
END_IF

(* Motor bekapcsolva *)
tMotorOn(IN:= (q_bConveyorOnL OR q_bConveyorOnR) AND NOT bError, 
	PT:= T#1S,
	Q=>  bMotorOn);

(* Manual reset *)
IF bError AND bAck AND NOT q_bConveyorRst THEN
	q_bConveyorRst := TRUE;
END_IF

tReset(IN:= q_bConveyorRst, PT:= timReset, Q=> , ET=> );
IF tReset.Q THEN
	q_bConveyorRst := FALSE;
END_IF

(*Hiba string*)
IF bErrOn OR bErrRun THEN
	sError := sName;
	IF bErrOn THEN
		sError :=  CONCAT(sError, aErrorDesc[0]);
	END_IF
	IF bErrRun THEN
		sError :=  CONCAT(sError, aErrorDesc[1]);
	END_IF
ELSE
	sError := sEmpty;
END_IF

(*Hiba kezelés Tc3_EventLogger*)
IF NOT bIsInitalized THEN
	bIsInitalized := TRUE;
	fbStartAlarm.CreateEx(stStartEvent, TRUE, 0);
	fbRunAlarm.CreateEx(stRunEvent, TRUE, 0);
END_IF

(*Hiba törlés (nyugtázott és megszűnt)*)
IF fbStartAlarm.eConfirmationState = 3 AND NOT bError THEN
	fbStartAlarm.Clear(0, FALSE);
END_IF	
IF fbRunAlarm.eConfirmationState = 3 AND NOT bError THEN
	fbRunAlarm.Clear(0, FALSE);
END_IF

END_FUNCTION_BLOCK

// ---- POUs/FBs/FB_BISL.TcPOU
FUNCTION_BLOCK FB_BISL
(*Ez az FB BIS L-409-045-001-07-SA olvasóval lett tezstelve
TAG: BIS003R BIS L-200-03/L, ami 40bit adatot ad vissza*)

VAR_INPUT
	sName				:STRING;
	KA					:BOOL; (*Head off=1/Head on = 0*)
	GR					:BOOL; (*SW Reset = 1 / Normal operation =0*)
	InData	AT %I*		:ARRAY[0..8] OF BYTE;
END_VAR
VAR_OUTPUT
	BB					:BOOL; (*Device ready=1 / Device in groung state =0*)
	HF					:BOOL; (*Head is turned off=1/turned on =0*)
	AF					:BOOL; (*Job incorrectly processed = 1 / without error = 0*)
	CP					:BOOL; (*Data carrier is within range of the head =1 / no data carrier = 0*)
	ErrorCode			:BYTE; (*Error codem when AF=1*)
	TAGData				:ULINT; (*Data wich were read from the data carrier*)
	OutData		AT %Q*	:ARRAY[0..7] OF BYTE;
END_VAR
VAR
END_VAR

BB:=InData[0].7;
HF:=InData[0].6;
AF:=InData[0].3;
CP:=InData[0].0;

IF AF
	THEN ErrorCode:=InData[1];
		 TAGData:=0;
	ELSE ErrorCode:=0;
		 IF CP
			 THEN TAGData:=
					SHL(BYTE_TO_ULINT(InData[8] AND 127), 56) +
					SHL(BYTE_TO_ULINT(InData[7]), 48) +
					SHL(BYTE_TO_ULINT(InData[6]), 40) +
					SHL(BYTE_TO_ULINT(InData[5]), 32) +
					SHL(BYTE_TO_ULINT(InData[4]), 24) +
					SHL(BYTE_TO_ULINT(InData[3]), 16) +
					SHL(BYTE_TO_ULINT(InData[2]), 8) +
					InData[1]; 
		 END_IF;
END_IF;
		 
OutData[0].2:=GR;
OutData[0].5:=KA;
OutData[7]:=OutData[0];

END_FUNCTION_BLOCK

// ---- POUs/FBs/FB_UserLed.TcPOU
FUNCTION_BLOCK FB_UserLed
VAR_INPUT
	bEnable					:BOOL;					// FB Engedély.
	eULedColor				:E_UsrLED_Color;
END_VAR
VAR_OUTPUT
	bError					:BOOL;					// Hiba bit
	nErrId					:UDINT;					// Hiba kód
END_VAR
VAR
	fbUserLED				:FB_SetLedColor_BAPI;
END_VAR

(*-----=== User LED ===-----*)
(*	--------------------------------------------------------------------------------
	Leírás		:	C69XX CPU User LED kezelés
	Név			:	FB_UserLed
	Módosító	:	Závori Zsolt
	Dátum		:	2019.07.05
	Revízió		:	1.0
	--------------------------------------------------------------------------------
	Feltételek	:	Tc2_IoFunctions
	Változók	:	-
	Visu		:	-
	UserControl	:	-
	--------------------------------------------------------------------------------
	Részletek	:	-					
*)
IF		fbUserLED.eNewColor <> eULedColor AND
		NOT fbUserLED.bExecute AND
		NOT fbUserLED.bBusy THEN
			fbUserLED.eNewColor := eULedColor;
			fbUserLED.bExecute := TRUE;
ELSIF	(fbUserLED.bExecute AND NOT fbUserLED.bBusy) OR fbUserLED.bError THEN
			fbUserLED.bExecute := FALSE;
END_IF
fbUserLED();
bError := fbUserLED.bError;
nErrId := fbUserLED.nErrID;

END_FUNCTION_BLOCK
